TYPE ST_INPUTS_BagFilters:
STRUCT
	
	Filter1_MaxDiffPressure:    UINT;
	Filter2_MaxDiffPressure:    UINT;

END_STRUCT
END_TYPE

(* stored: Version 1.1.0.1, ProductVersion 3.1.4024.12
   DUT ST_INPUTS_BagFilters: Id {cc839e59-5a4b-47bd-8dbe-02a13eae3cac} *)
